{attribute addProperty BoxType "EP4378-1022-0017"}
{attribute addProperty Id "OutputAT %Q*BOOL81"}
{attribute addProperty CRC "2134331056"}
{attribute addProperty SizeInBites "8"}
{attribute addProperty SizeInBytes "1"}
TYPE DO_X08_Pin4_Output_7F374EB0 :
STRUCT
	{attribute addProperty Name "Output"}
	Output AT %Q* : BOOL;
END_STRUCT
END_TYPE

(* stored: Version 1.2.0.0, ProductVersion 3.1.4024.9
   DUT DO_X08_Pin4_Output_7F374EB0: Id {9ebb74f0-b172-42cc-8d5c-7a961b8e29c1} *)
